(* IEC 61131-3 sources: automatic-screwdriver-line/src/POU/Interface, 7 files *)

(* ---- I_Actuator.st ---- *)
// Generated from Automatic_ScrewDriver_Line.xml by tools/export_st.py - do not edit.
// The CODESYS project is the source of truth.

INTERFACE I_Actuator

METHOD Enable : BOOL
END_METHOD

METHOD Disable : BOOL
END_METHOD

END_INTERFACE

(* ---- I_Device.st ---- *)
// Generated from Automatic_ScrewDriver_Line.xml by tools/export_st.py - do not edit.
// The CODESYS project is the source of truth.

INTERFACE I_Device EXTENDS I_Actuator

END_INTERFACE

(* ---- I_Diagnosable.st ---- *)
// Generated from Automatic_ScrewDriver_Line.xml by tools/export_st.py - do not edit.
// The CODESYS project is the source of truth.

INTERFACE I_Diagnosable

METHOD GetError : ErrorCode
END_METHOD

METHOD ClearError : BOOL
END_METHOD

END_INTERFACE

(* ---- I_Mover.st ---- *)
// Generated from Automatic_ScrewDriver_Line.xml by tools/export_st.py - do not edit.
// The CODESYS project is the source of truth.

INTERFACE I_Mover EXTENDS I_Device

METHOD MoveToPosition : BOOL
VAR_INPUT
	Position : REAL;
END_VAR
END_METHOD

END_INTERFACE

(* ---- I_ReportSink.st ---- *)
// Generated from Automatic_ScrewDriver_Line.xml by tools/export_st.py - do not edit.
// The CODESYS project is the source of truth.

INTERFACE I_ReportSink

METHOD PublishReport : BOOL
VAR_INPUT
	Report : JobReport;
END_VAR
END_METHOD

END_INTERFACE

(* ---- I_Resettable.st ---- *)
// Generated from Automatic_ScrewDriver_Line.xml by tools/export_st.py - do not edit.
// The CODESYS project is the source of truth.

INTERFACE I_Resettable

METHOD Reset : BOOL
END_METHOD

END_INTERFACE

(* ---- I_Tool.st ---- *)
// Generated from Automatic_ScrewDriver_Line.xml by tools/export_st.py - do not edit.
// The CODESYS project is the source of truth.

INTERFACE I_Tool EXTENDS I_Device

METHOD ProcessTool : BOOL
VAR_INPUT
	Angle : DINT;
END_VAR
END_METHOD

END_INTERFACE
